// SIMATIC S7-200 project (STEP 7-Micro/WIN), CPU 224 REL 02.01

ORGANIZATION_BLOCK MAIN:OB1
TITLE=PROGRAM COMMENTS
BEGIN
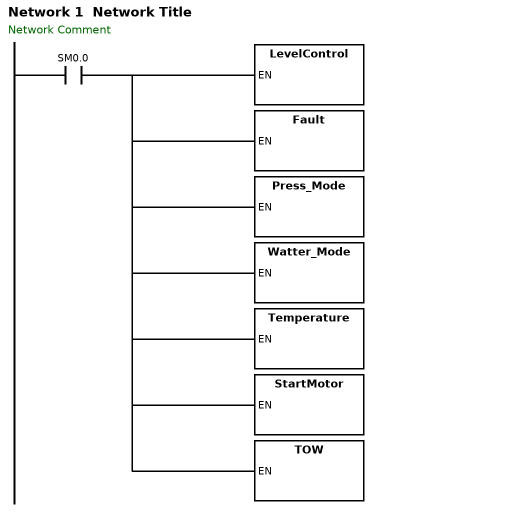
Network 1 // Network Title
// Network Comment
LD     SM0.0
CALL   LevelControl:SBR0
CALL   Fault:SBR1
CALL   Press_Mode:SBR2
CALL   Watter_Mode:SBR3
CALL   Temperature:SBR4
CALL   StartMotor:SBR5
CALL   TOW:SBR6
END_ORGANIZATION_BLOCK

SUBROUTINE_BLOCK LevelControl:SBR0
TITLE=SUBROUTINE COMMENTS
BEGIN
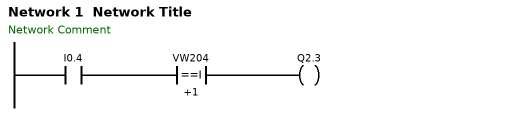
Network 1 // Network Title
// Network Comment
LD     I0.4
AW=    VW204, +1
=      Q2.3
END_SUBROUTINE_BLOCK

SUBROUTINE_BLOCK Fault:SBR1
TITLE=
BEGIN
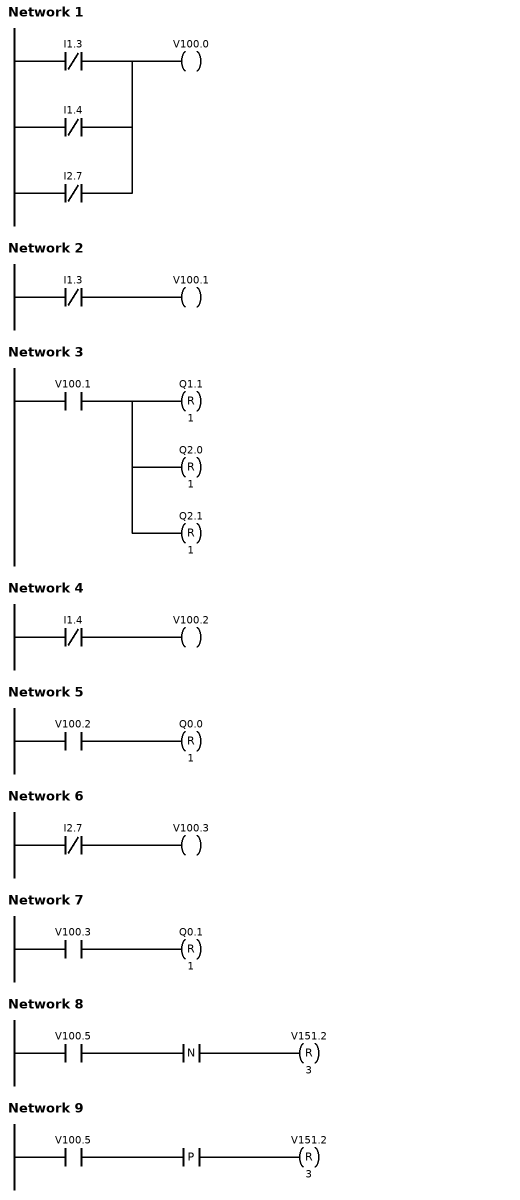
Network 1
LDN    I1.3
ON     I1.4
ON     I2.7
=      V100.0
Network 2
LDN    I1.3
=      V100.1
Network 3
LD     V100.1
R      Q1.1, 1
R      Q2.0, 1
R      Q2.1, 1
Network 4
LDN    I1.4
=      V100.2
Network 5
LD     V100.2
R      Q0.0, 1
Network 6
LDN    I2.7
=      V100.3
Network 7
LD     V100.3
R      Q0.1, 1
Network 8
LD     V100.5
ED
R      V151.2, 3
Network 9
LD     V100.5
EU
R      V151.2, 3
END_SUBROUTINE_BLOCK

SUBROUTINE_BLOCK Press_Mode:SBR2
TITLE=
BEGIN
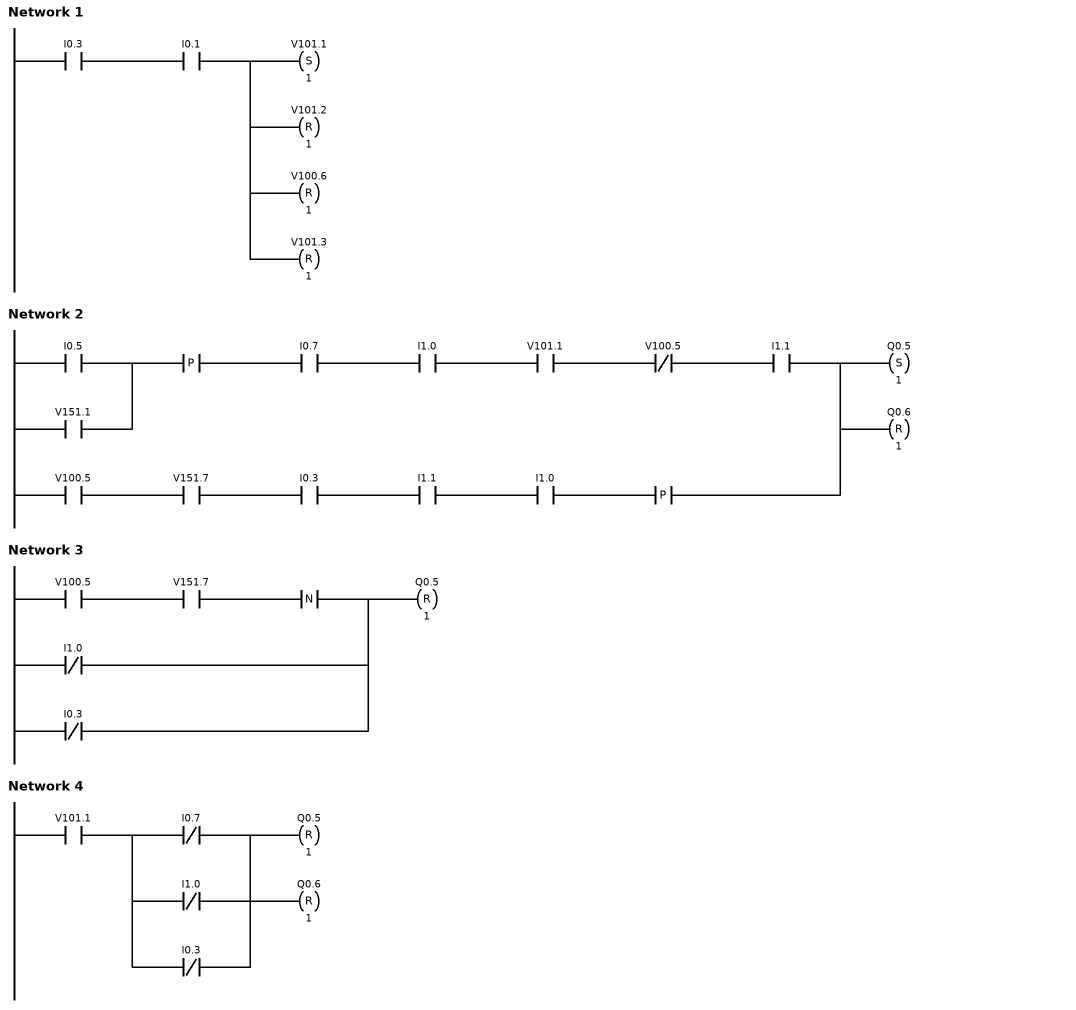
Network 1
LD     I0.3
A      I0.1
S      V101.1, 1
R      V101.2, 1
R      V100.6, 1
R      V101.3, 1
Network 2
LD     I0.5
O      V151.1
EU
A      I0.7
A      I1.0
A      V101.1
AN     V100.5
A      I1.1
LD     V100.5
A      V151.7
A      I0.3
A      I1.1
A      I1.0
EU
OLD
S      Q0.5, 1
R      Q0.6, 1
Network 3
LD     V100.5
A      V151.7
ED
ON     I1.0
ON     I0.3
R      Q0.5, 1
Network 4
LD     V101.1
LDN    I0.7
ON     I1.0
ON     I0.3
ALD
R      Q0.5, 1
R      Q0.6, 1
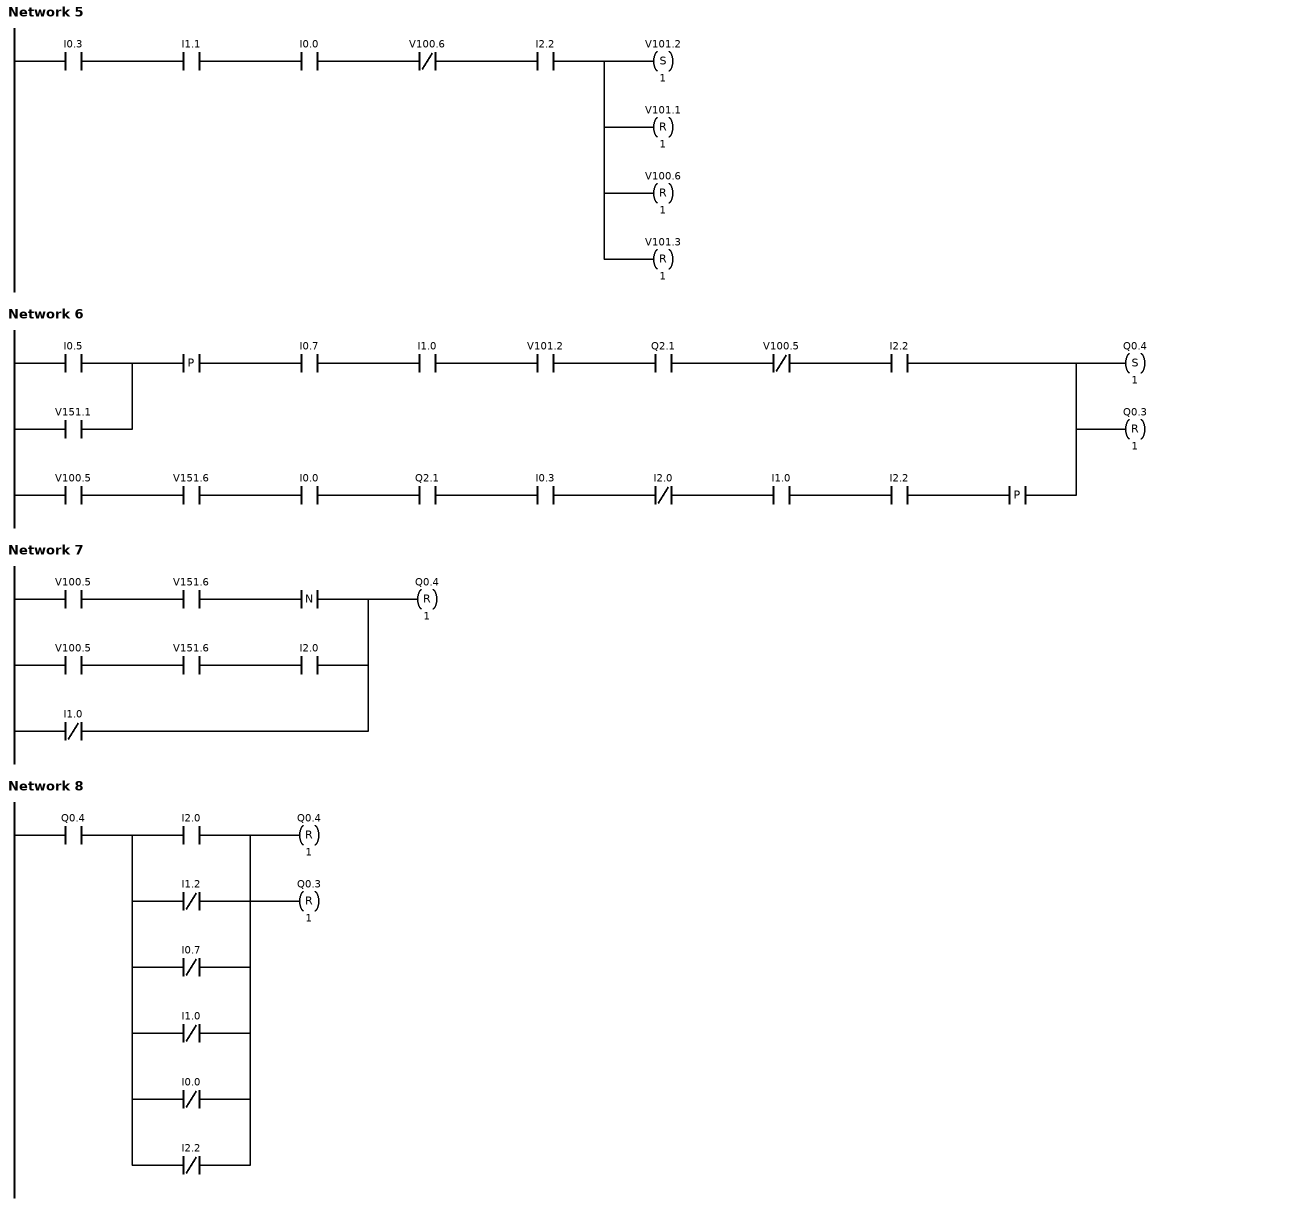
Network 5
LD     I0.3
A      I1.1
A      I0.0
AN     V100.6
A      I2.2
S      V101.2, 1
R      V101.1, 1
R      V100.6, 1
R      V101.3, 1
Network 6
LD     I0.5
O      V151.1
EU
A      I0.7
A      I1.0
A      V101.2
A      Q2.1
AN     V100.5
A      I2.2
LD     V100.5
A      V151.6
A      I0.0
A      Q2.1
A      I0.3
AN     I2.0
A      I1.0
A      I2.2
EU
OLD
S      Q0.4, 1
R      Q0.3, 1
Network 7
LD     V100.5
A      V151.6
ED
LD     V100.5
A      V151.6
A      I2.0
OLD
ON     I1.0
R      Q0.4, 1
Network 8
LD     Q0.4
LD     I2.0
ON     I1.2
ON     I0.7
ON     I1.0
ON     I0.0
ON     I2.2
ALD
R      Q0.4, 1
R      Q0.3, 1
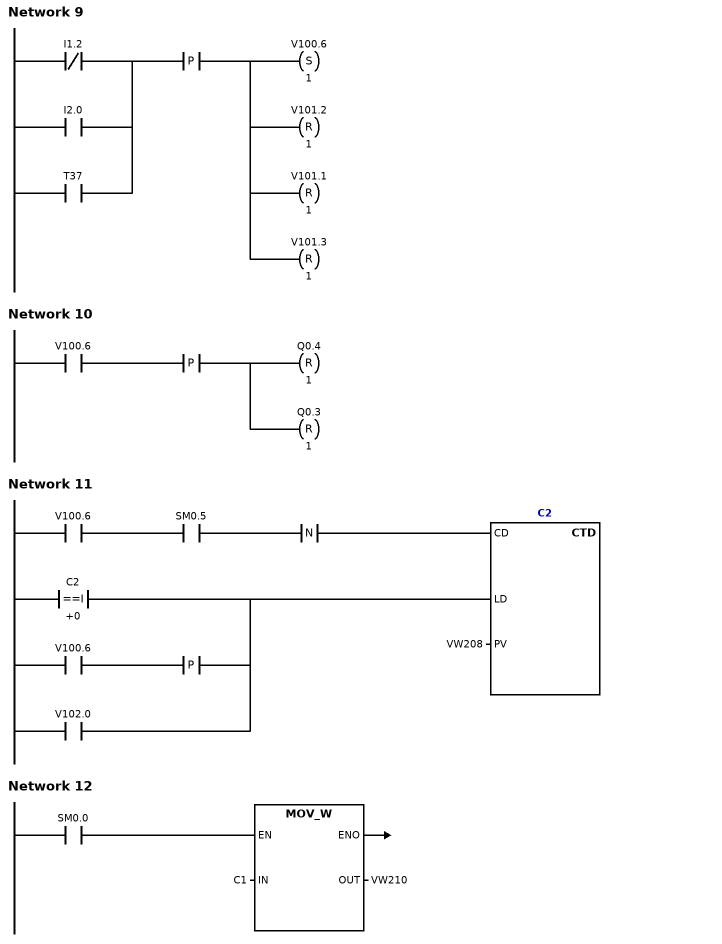
Network 9
LDN    I1.2
O      I2.0
O      T37
EU
S      V100.6, 1
R      V101.2, 1
R      V101.1, 1
R      V101.3, 1
Network 10
LD     V100.6
EU
R      Q0.4, 1
R      Q0.3, 1
Network 11
LD     V100.6
A      SM0.5
ED
LDW=   C2, +0
LD     V100.6
EU
OLD
O      V102.0
CTD    C2, VW208
Network 12
LD     SM0.0
MOVW   C1, VW210
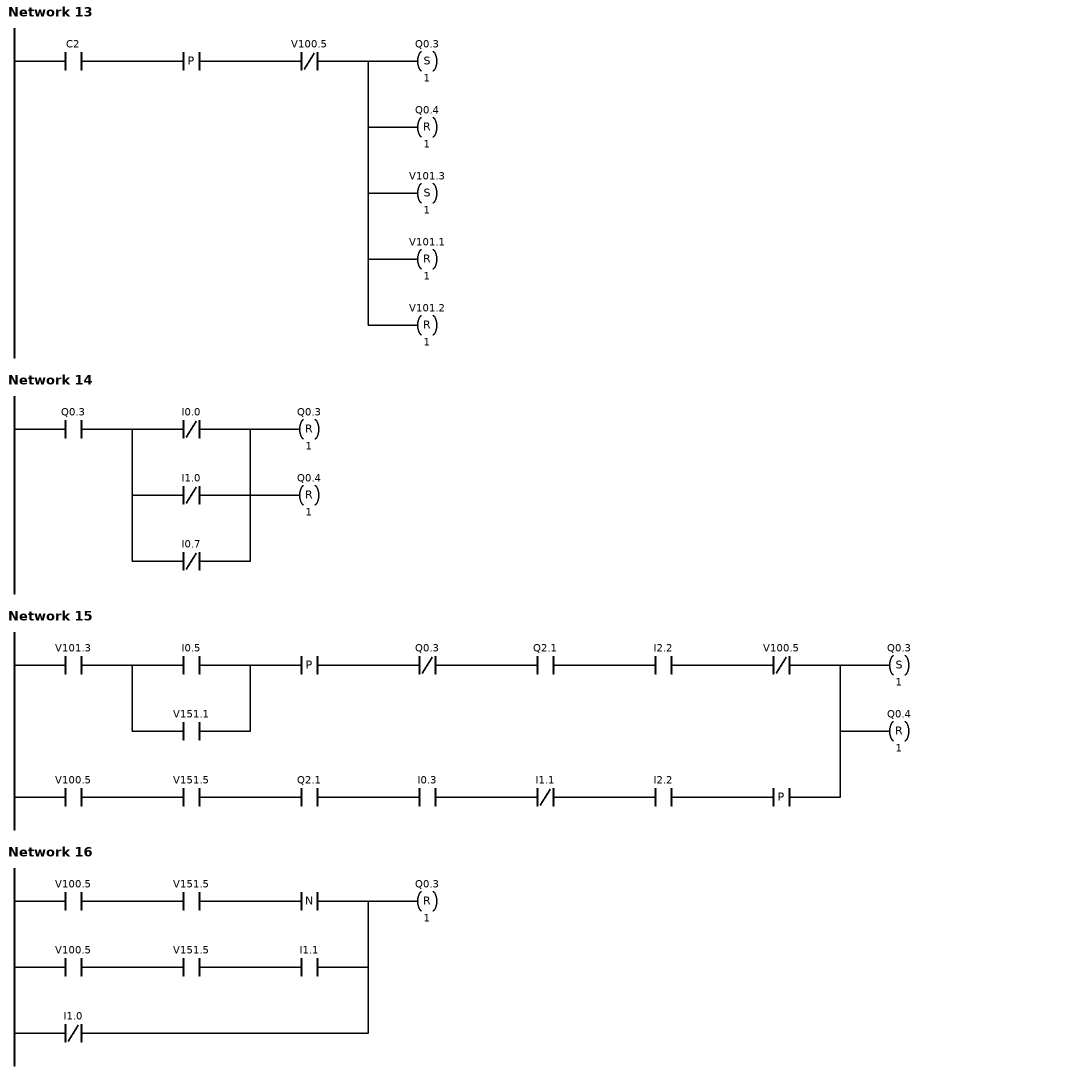
Network 13
LD     C2
EU
AN     V100.5
S      Q0.3, 1
R      Q0.4, 1
S      V101.3, 1
R      V101.1, 1
R      V101.2, 1
Network 14
LD     Q0.3
LDN    I0.0
ON     I1.0
ON     I0.7
ALD
R      Q0.3, 1
R      Q0.4, 1
Network 15
LD     V101.3
LD     I0.5
O      V151.1
ALD
EU
AN     Q0.3
A      Q2.1
A      I2.2
AN     V100.5
LD     V100.5
A      V151.5
A      Q2.1
A      I0.3
AN     I1.1
A      I2.2
EU
OLD
S      Q0.3, 1
R      Q0.4, 1
Network 16
LD     V100.5
A      V151.5
ED
LD     V100.5
A      V151.5
A      I1.1
OLD
ON     I1.0
R      Q0.3, 1
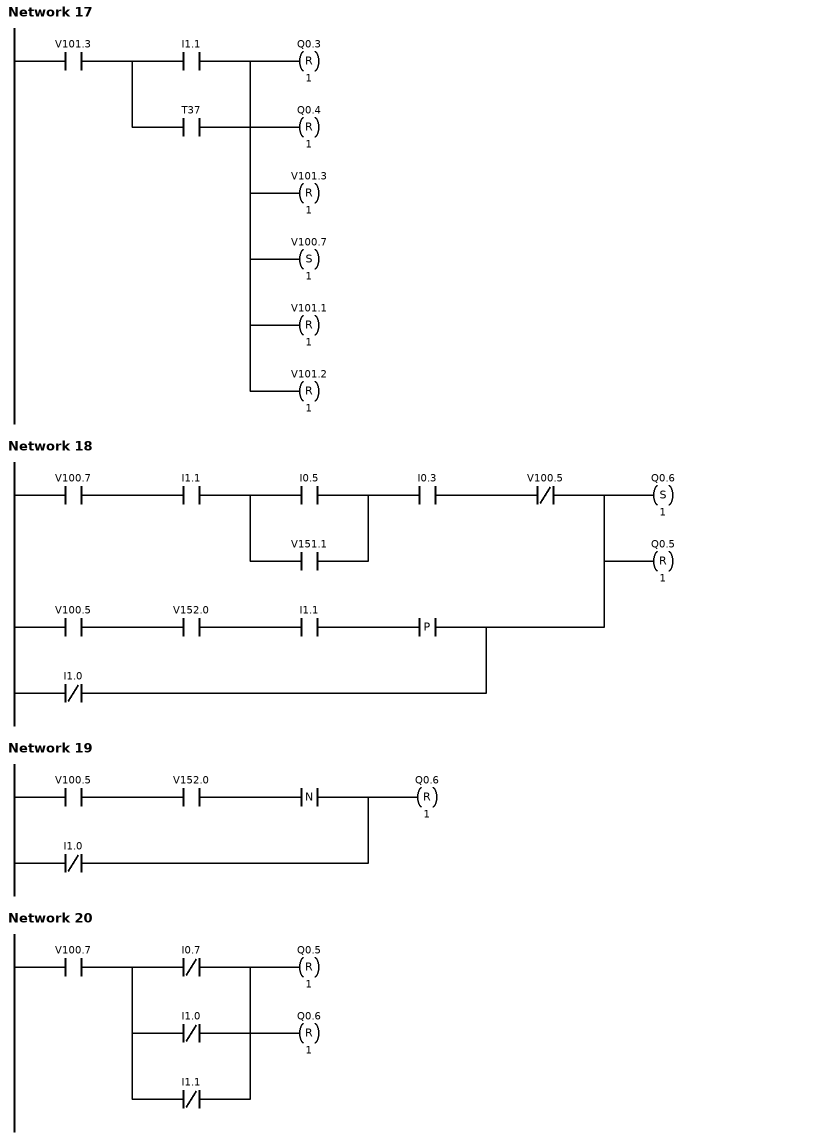
Network 17
LD     V101.3
LD     I1.1
O      T37
ALD
R      Q0.3, 1
R      Q0.4, 1
R      V101.3, 1
S      V100.7, 1
R      V101.1, 1
R      V101.2, 1
Network 18
LD     V100.7
A      I1.1
LD     I0.5
O      V151.1
ALD
A      I0.3
AN     V100.5
LD     V100.5
A      V152.0
A      I1.1
EU
ON     I1.0
OLD
S      Q0.6, 1
R      Q0.5, 1
Network 19
LD     V100.5
A      V152.0
ED
ON     I1.0
R      Q0.6, 1
Network 20
LD     V100.7
LDN    I0.7
ON     I1.0
ON     I1.1
ALD
R      Q0.5, 1
R      Q0.6, 1
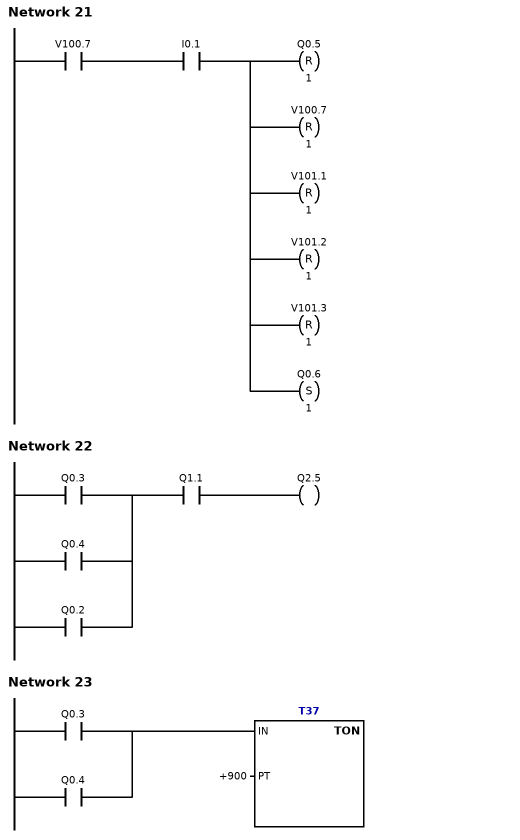
Network 21
LD     V100.7
A      I0.1
R      Q0.5, 1
R      V100.7, 1
R      V101.1, 1
R      V101.2, 1
R      V101.3, 1
S      Q0.6, 1
Network 22
LD     Q0.3
O      Q0.4
O      Q0.2
A      Q1.1
=      Q2.5
Network 23
LD     Q0.3
O      Q0.4
TON    T37, +900
END_SUBROUTINE_BLOCK

SUBROUTINE_BLOCK Watter_Mode:SBR3
TITLE=
BEGIN
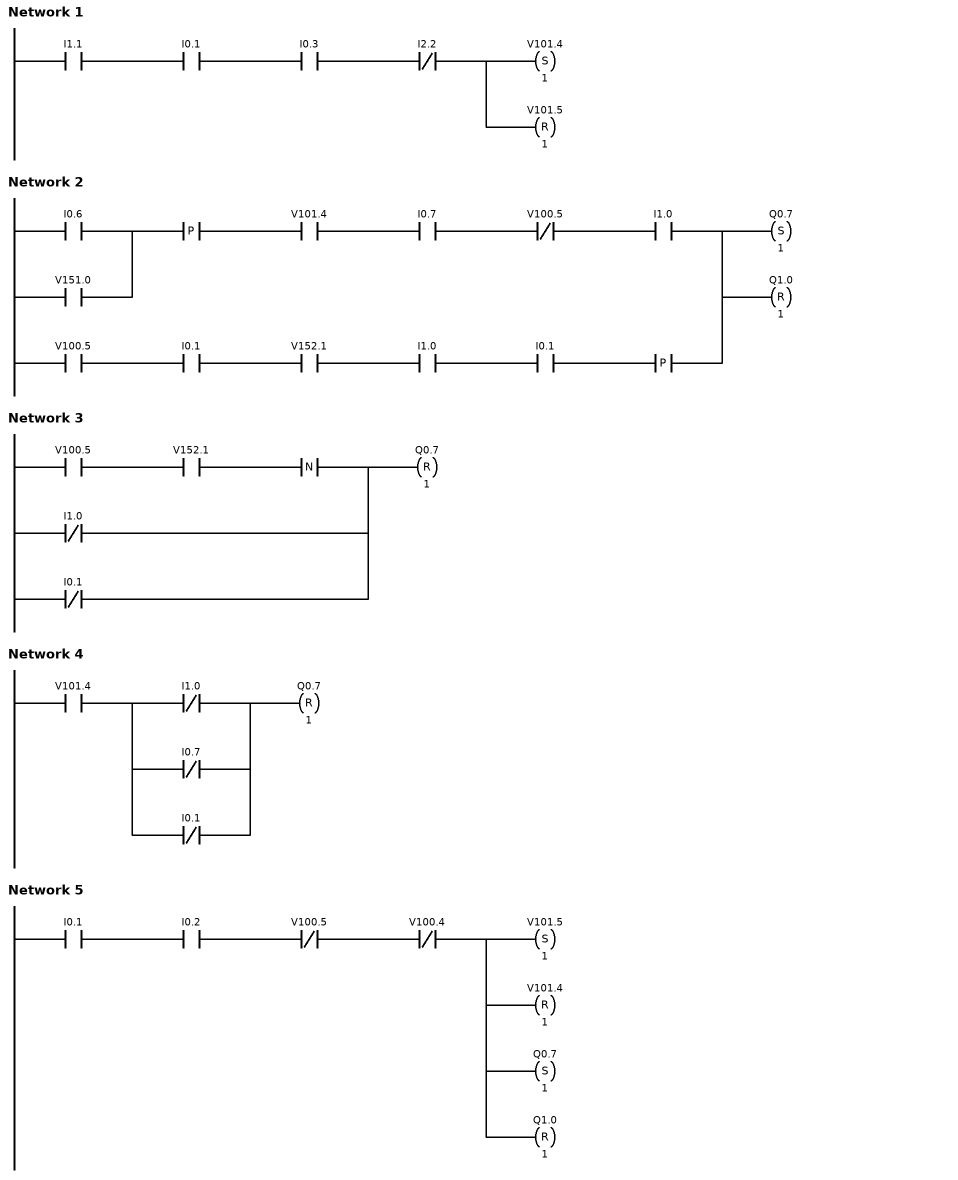
Network 1
LD     I1.1
A      I0.1
A      I0.3
AN     I2.2
S      V101.4, 1
R      V101.5, 1
Network 2
LD     I0.6
O      V151.0
EU
A      V101.4
A      I0.7
AN     V100.5
A      I1.0
LD     V100.5
A      I0.1
A      V152.1
A      I1.0
A      I0.1
EU
OLD
S      Q0.7, 1
R      Q1.0, 1
Network 3
LD     V100.5
A      V152.1
ED
ON     I1.0
ON     I0.1
R      Q0.7, 1
Network 4
LD     V101.4
LDN    I1.0
ON     I0.7
ON     I0.1
ALD
R      Q0.7, 1
Network 5
LD     I0.1
A      I0.2
AN     V100.5
AN     V100.4
S      V101.5, 1
R      V101.4, 1
S      Q0.7, 1
R      Q1.0, 1
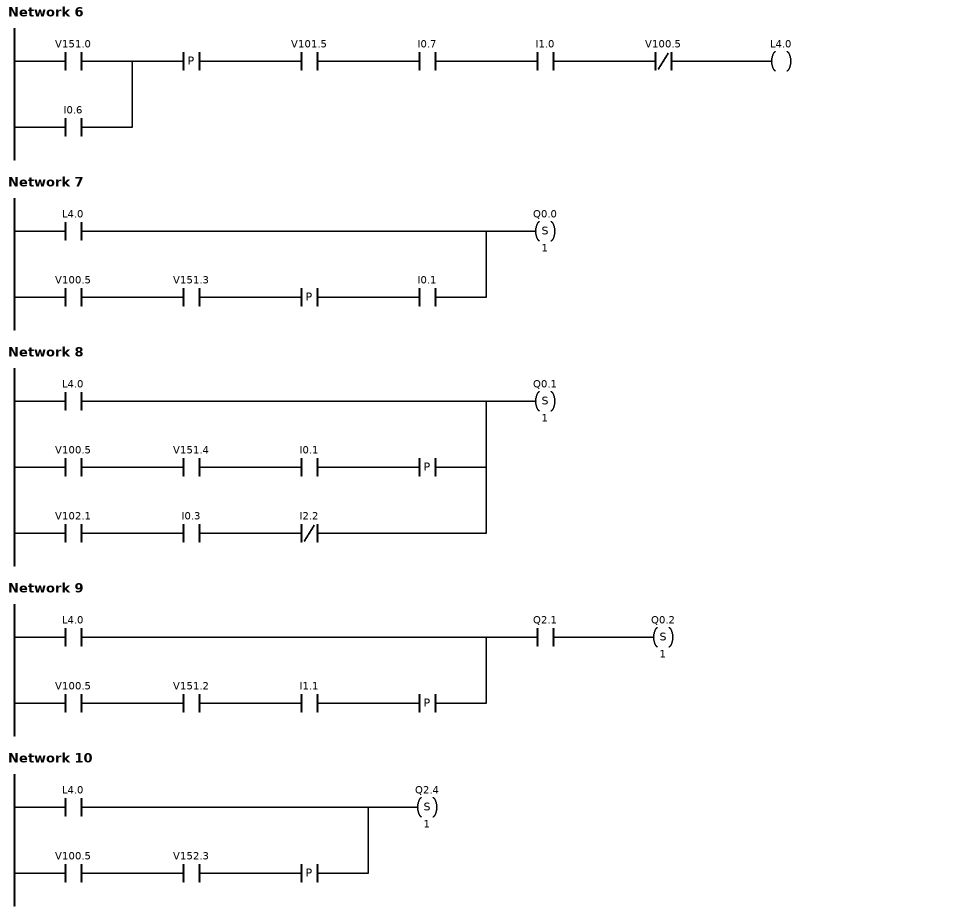
Network 6
LD     V151.0
O      I0.6
EU
A      V101.5
A      I0.7
A      I1.0
AN     V100.5
=      L4.0
Network 7
LD     L4.0
LD     V100.5
A      V151.3
EU
A      I0.1
OLD
S      Q0.0, 1
Network 8
LD     L4.0
LD     V100.5
A      V151.4
A      I0.1
EU
OLD
LD     V102.1
A      I0.3
AN     I2.2
OLD
S      Q0.1, 1
Network 9
LD     L4.0
LD     V100.5
A      V151.2
A      I1.1
EU
OLD
A      Q2.1
S      Q0.2, 1
Network 10
LD     L4.0
LD     V100.5
A      V152.3
EU
OLD
S      Q2.4, 1
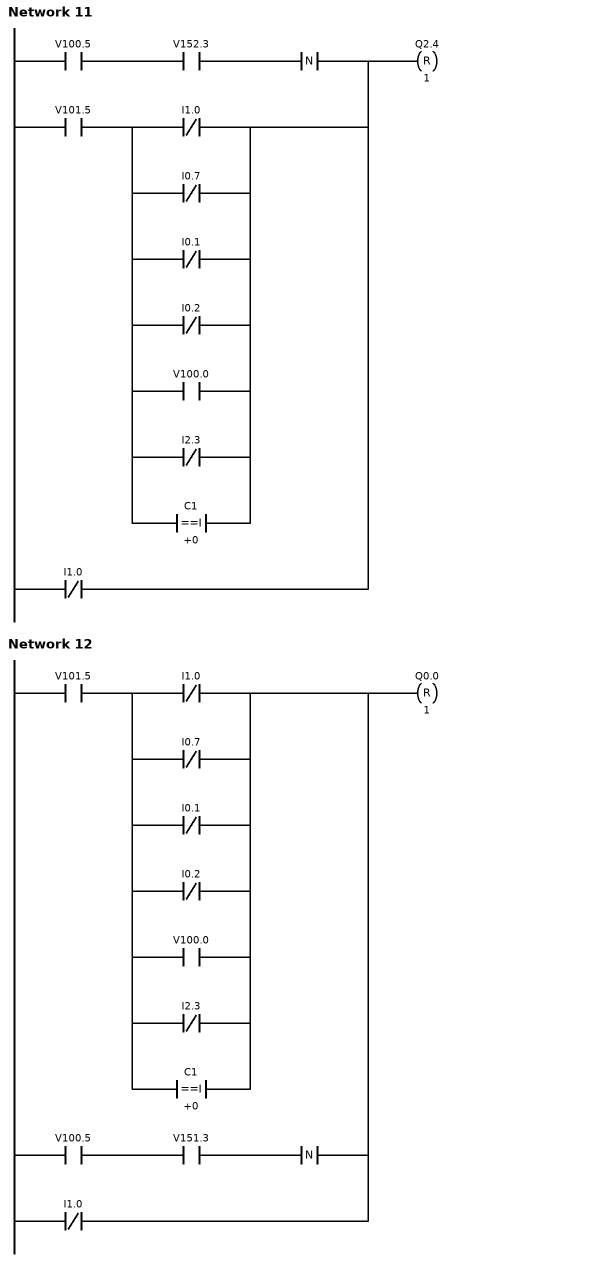
Network 11
LD     V100.5
A      V152.3
ED
LD     V101.5
LDN    I1.0
ON     I0.7
ON     I0.1
ON     I0.2
O      V100.0
ON     I2.3
OW=    C1, +0
ALD
OLD
ON     I1.0
R      Q2.4, 1
Network 12
LD     V101.5
LDN    I1.0
ON     I0.7
ON     I0.1
ON     I0.2
O      V100.0
ON     I2.3
OW=    C1, +0
ALD
LD     V100.5
A      V151.3
ED
ON     I1.0
OLD
R      Q0.0, 1
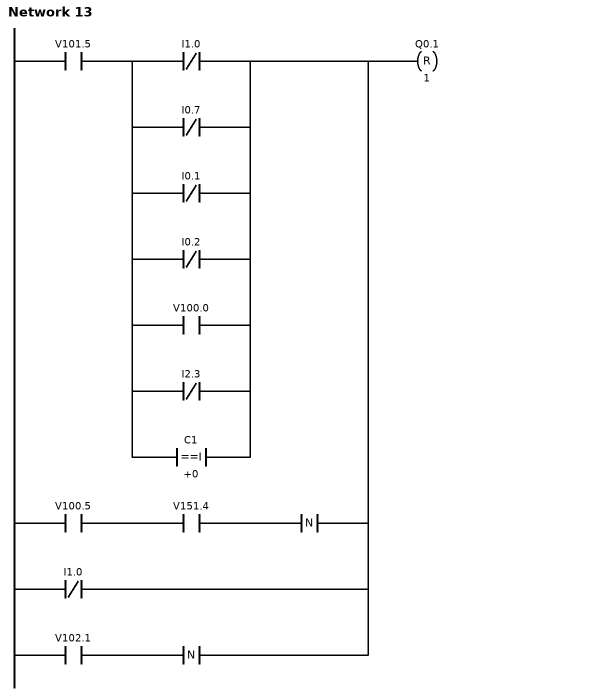
Network 13
LD     V101.5
LDN    I1.0
ON     I0.7
ON     I0.1
ON     I0.2
O      V100.0
ON     I2.3
OW=    C1, +0
ALD
LD     V100.5
A      V151.4
ED
ON     I1.0
LD     V102.1
ED
OLD
OLD
R      Q0.1, 1
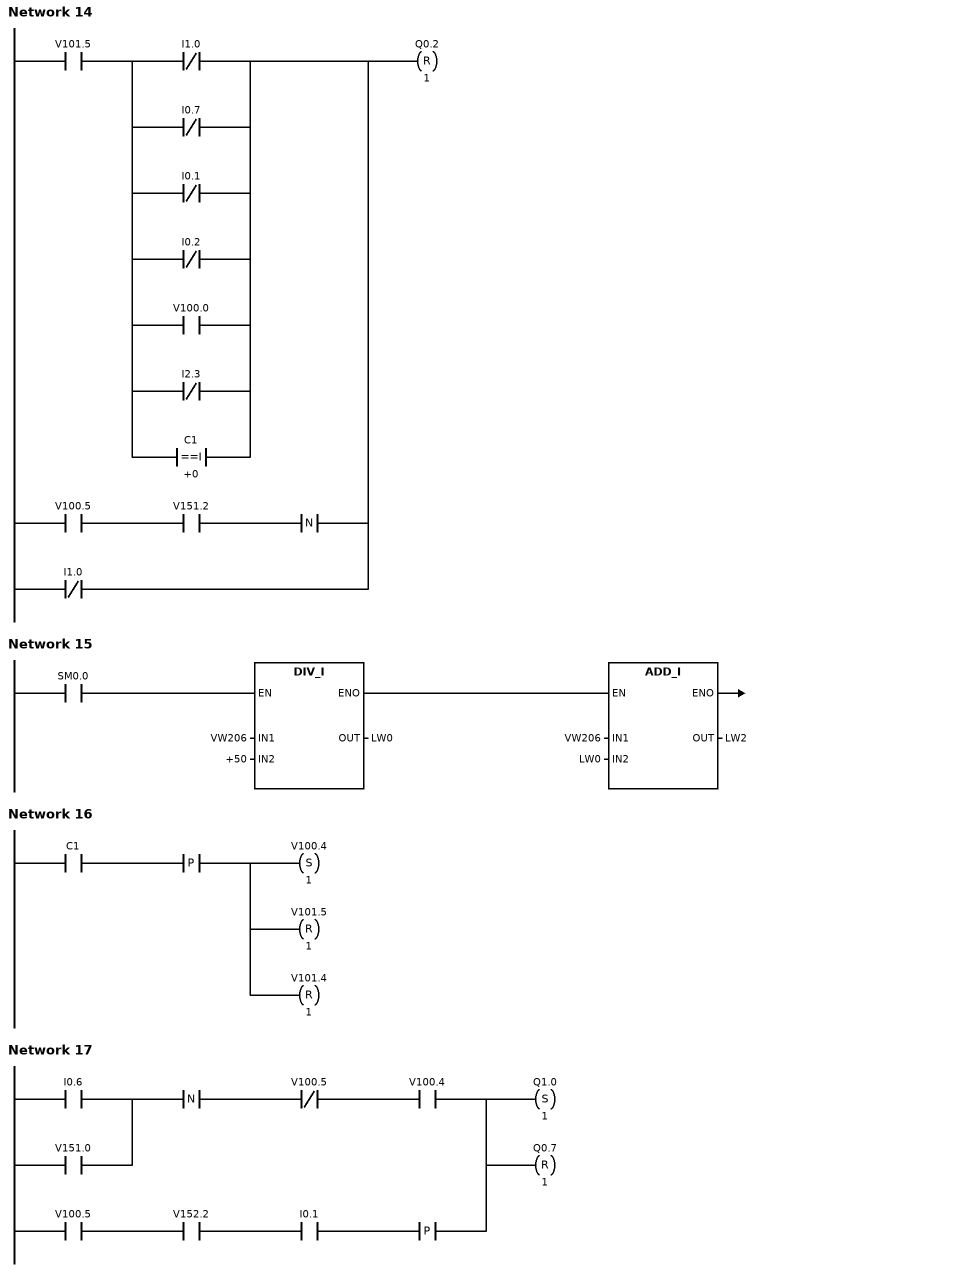
Network 14
LD     V101.5
LDN    I1.0
ON     I0.7
ON     I0.1
ON     I0.2
O      V100.0
ON     I2.3
OW=    C1, +0
ALD
LD     V100.5
A      V151.2
ED
ON     I1.0
OLD
R      Q0.2, 1
Network 15
LD     SM0.0
MOVW   VW206, LW0
AENO
/I     +50, LW0
AENO
MOVW   VW206, LW2
+I     LW0, LW2
Network 16
LD     C1
EU
S      V100.4, 1
R      V101.5, 1
R      V101.4, 1
Network 17
LD     I0.6
O      V151.0
ED
AN     V100.5
A      V100.4
LD     V100.5
A      V152.2
A      I0.1
EU
OLD
S      Q1.0, 1
R      Q0.7, 1
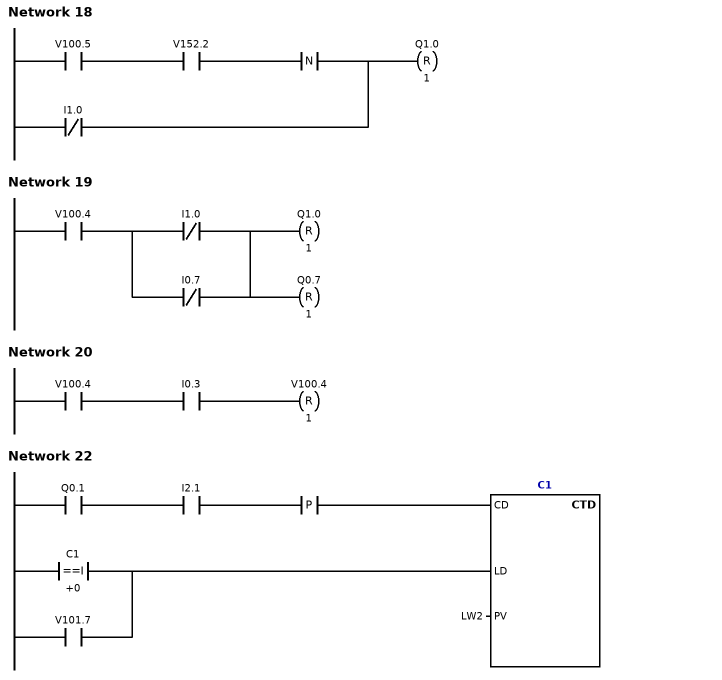
Network 18
LD     V100.5
A      V152.2
ED
ON     I1.0
R      Q1.0, 1
Network 19
LD     V100.4
LDN    I1.0
ON     I0.7
ALD
R      Q1.0, 1
R      Q0.7, 1
Network 20
LD     V100.4
A      I0.3
R      V100.4, 1
Network 22
LD     Q0.1
A      I2.1
EU
LDW=   C1, +0
O      V101.7
CTD    C1, LW2
END_SUBROUTINE_BLOCK

SUBROUTINE_BLOCK Temperature:SBR4
TITLE=
BEGIN
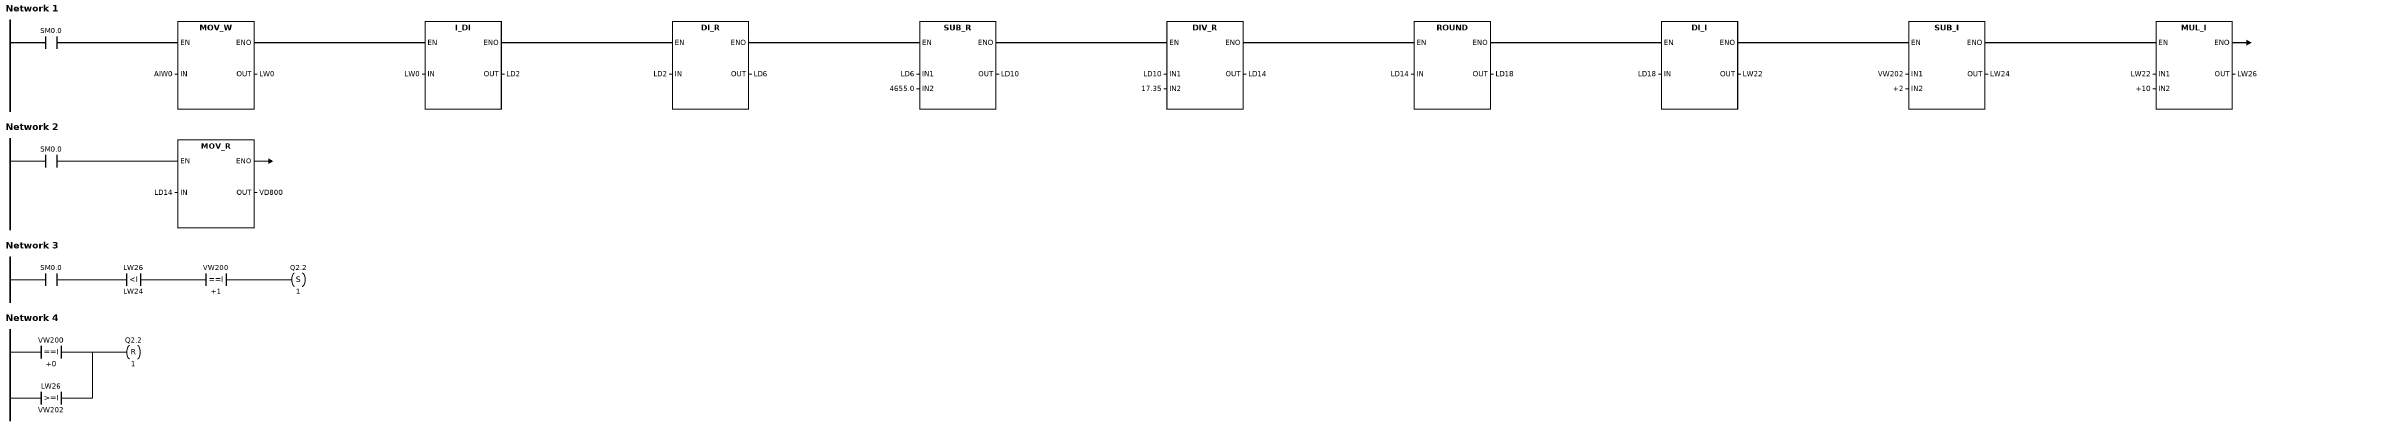
Network 1
LD     SM0.0
MOVW   AIW0, LW0
AENO
ITD    LW0, LD2
AENO
DTR    LD2, LD6
AENO
MOVR   LD6, LD10
AENO
-R     4655.0, LD10
AENO
MOVR   LD10, LD14
AENO
/R     17.35, LD14
AENO
ROUND  LD14, LD18
AENO
DTI    LD18, LW22
AENO
MOVW   VW202, LW24
AENO
-I     +2, LW24
AENO
MOVW   LW22, LW26
*I     +10, LW26
Network 2
LD     SM0.0
MOVR   LD14, VD800
Network 3
LD     SM0.0
AW<    LW26, LW24
AW=    VW200, +1
S      Q2.2, 1
Network 4
LDW=   VW200, +0
OW>=   LW26, VW202
R      Q2.2, 1
END_SUBROUTINE_BLOCK

SUBROUTINE_BLOCK StartMotor:SBR5
TITLE=
BEGIN
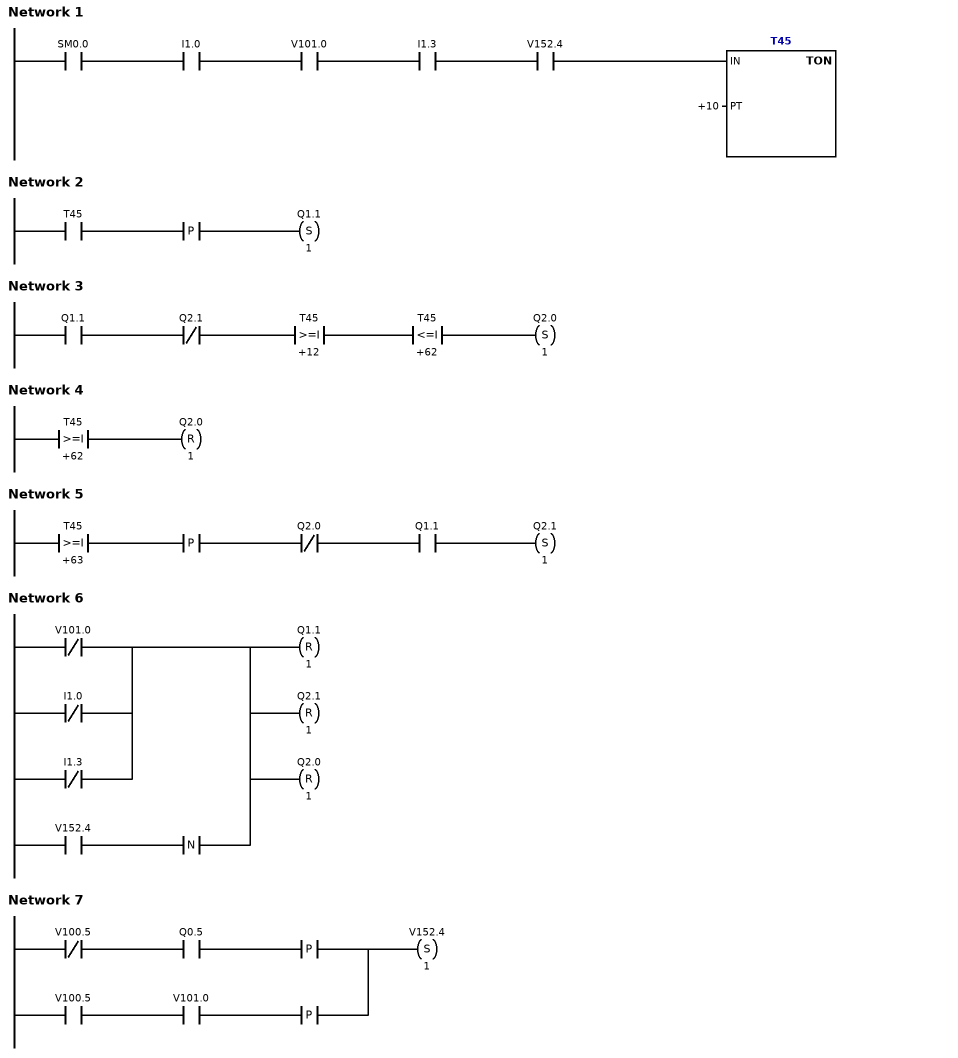
Network 1
LD     SM0.0
A      I1.0
A      V101.0
A      I1.3
A      V152.4
TON    T45, +10
Network 2
LD     T45
EU
S      Q1.1, 1
Network 3
LD     Q1.1
AN     Q2.1
AW>=   T45, +12
AW<=   T45, +62
S      Q2.0, 1
Network 4
LDW>=  T45, +62
R      Q2.0, 1
Network 5
LDW>=  T45, +63
EU
AN     Q2.0
A      Q1.1
S      Q2.1, 1
Network 6
LDN    V101.0
ON     I1.0
ON     I1.3
LD     V152.4
ED
OLD
R      Q1.1, 1
R      Q2.1, 1
R      Q2.0, 1
Network 7
LDN    V100.5
A      Q0.5
EU
LD     V100.5
A      V101.0
EU
OLD
S      V152.4, 1
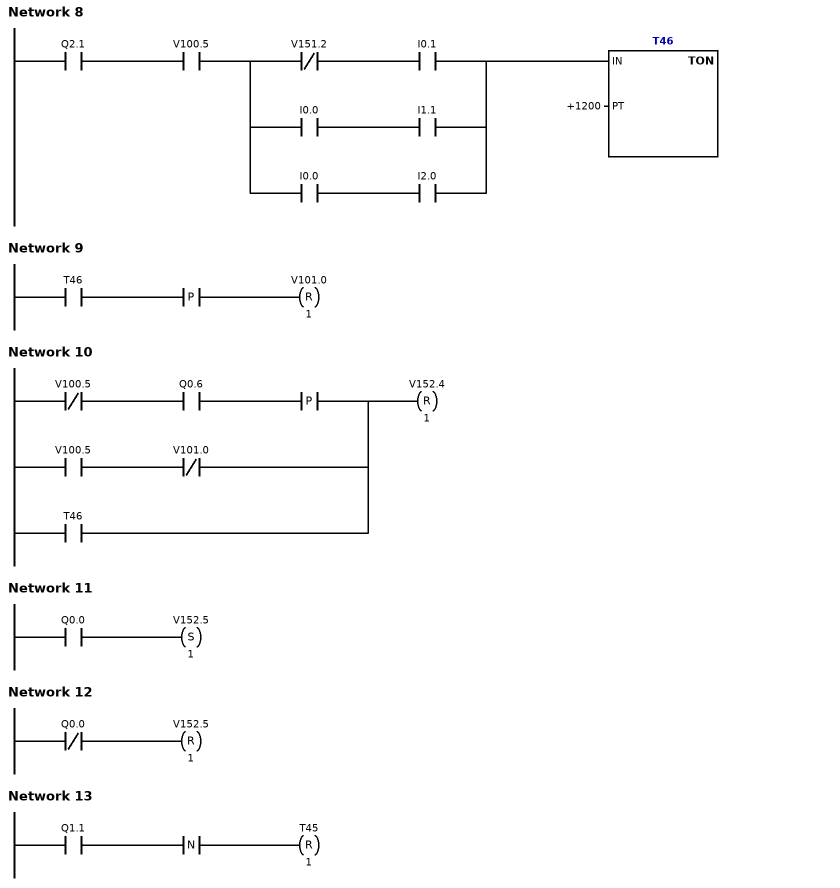
Network 8
LD     Q2.1
A      V100.5
LDN    V151.2
A      I0.1
LD     I0.0
A      I1.1
OLD
LD     I0.0
A      I2.0
OLD
ALD
TON    T46, +1200
Network 9
LD     T46
EU
R      V101.0, 1
Network 10
LDN    V100.5
A      Q0.6
EU
LD     V100.5
AN     V101.0
OLD
O      T46
R      V152.4, 1
Network 11
LD     Q0.0
S      V152.5, 1
Network 12
LDN    Q0.0
R      V152.5, 1
Network 13
LD     Q1.1
ED
R      T45, 1
END_SUBROUTINE_BLOCK

SUBROUTINE_BLOCK TOW:SBR6
TITLE=
BEGIN
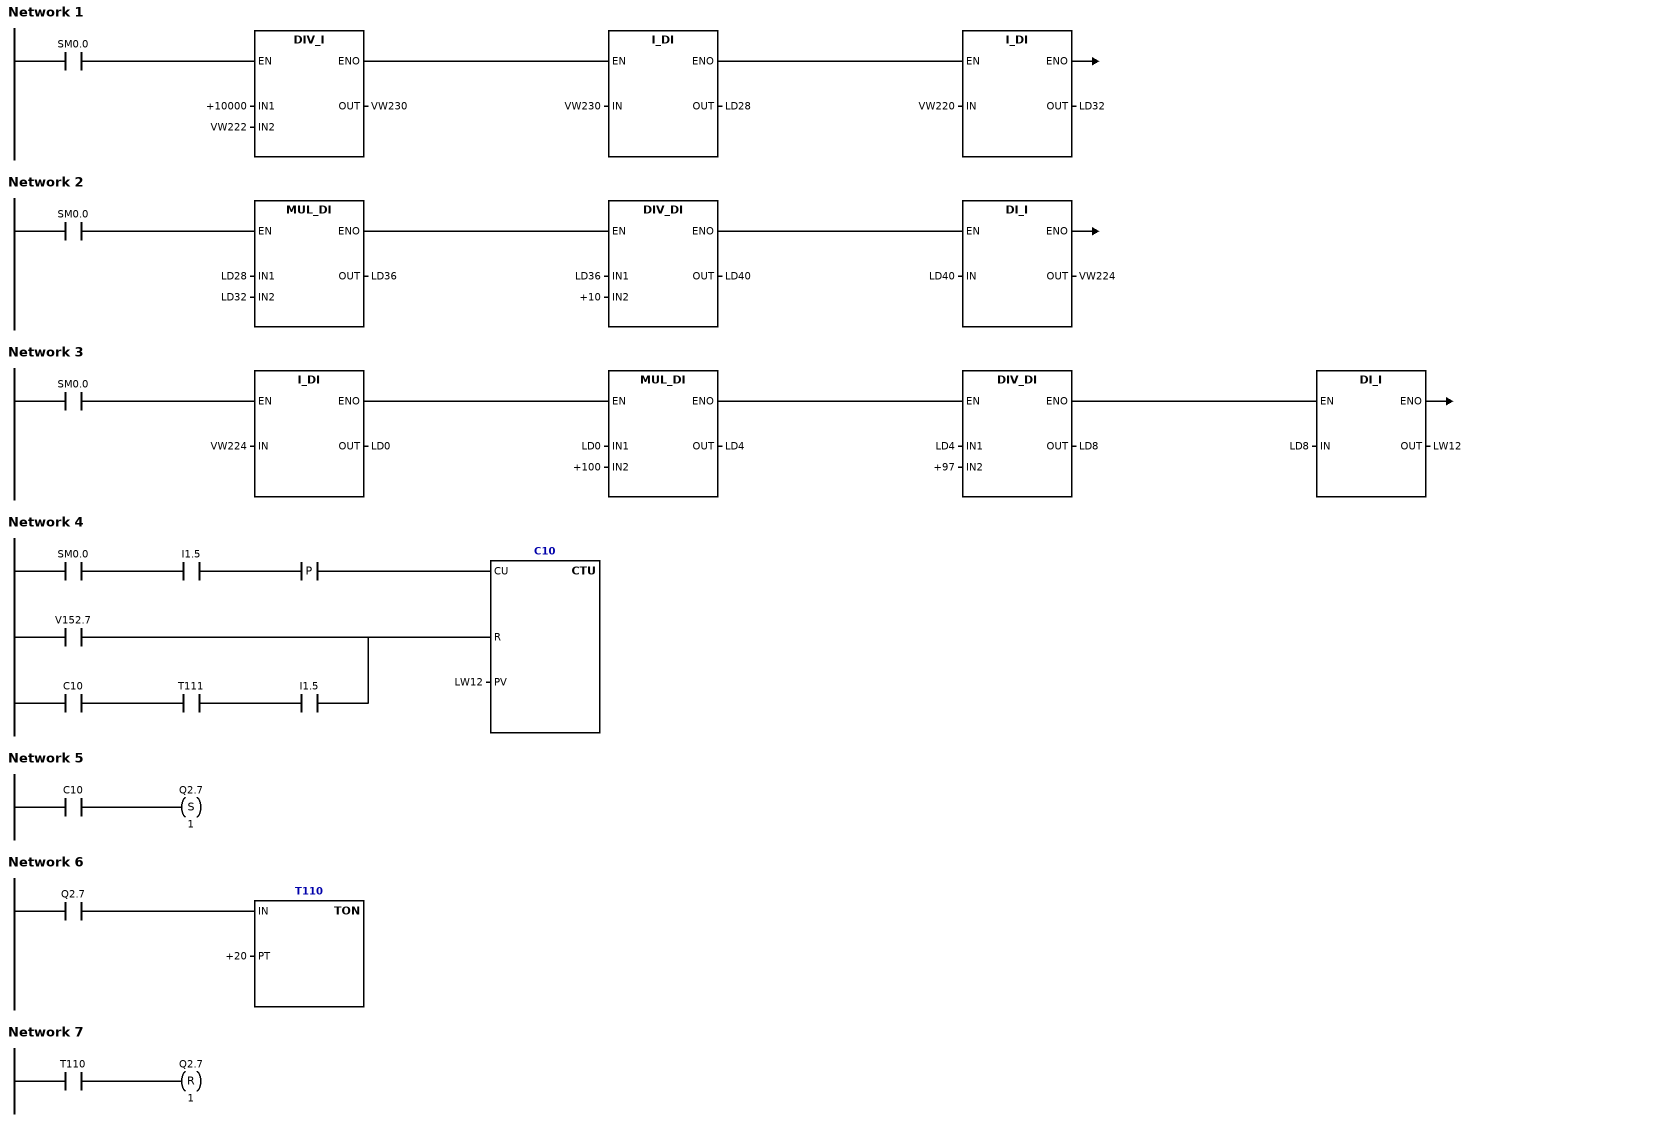
Network 1
LD     SM0.0
MOVW   +10000, VW230
AENO
/I     VW222, VW230
AENO
ITD    VW230, LD28
AENO
ITD    VW220, LD32
Network 2
LD     SM0.0
MOVD   LD28, LD36
AENO
*D     LD32, LD36
AENO
MOVD   LD36, LD40
AENO
/D     +10, LD40
AENO
DTI    LD40, VW224
Network 3
LD     SM0.0
ITD    VW224, LD0
AENO
MOVD   LD0, LD4
AENO
*D     +100, LD4
AENO
MOVD   LD4, LD8
AENO
/D     +97, LD8
AENO
DTI    LD8, LW12
Network 4
LD     SM0.0
A      I1.5
EU
LD     V152.7
LD     C10
A      T111
A      I1.5
OLD
CTU    C10, LW12
Network 5
LD     C10
S      Q2.7, 1
Network 6
LD     Q2.7
TON    T110, +20
Network 7
LD     T110
R      Q2.7, 1
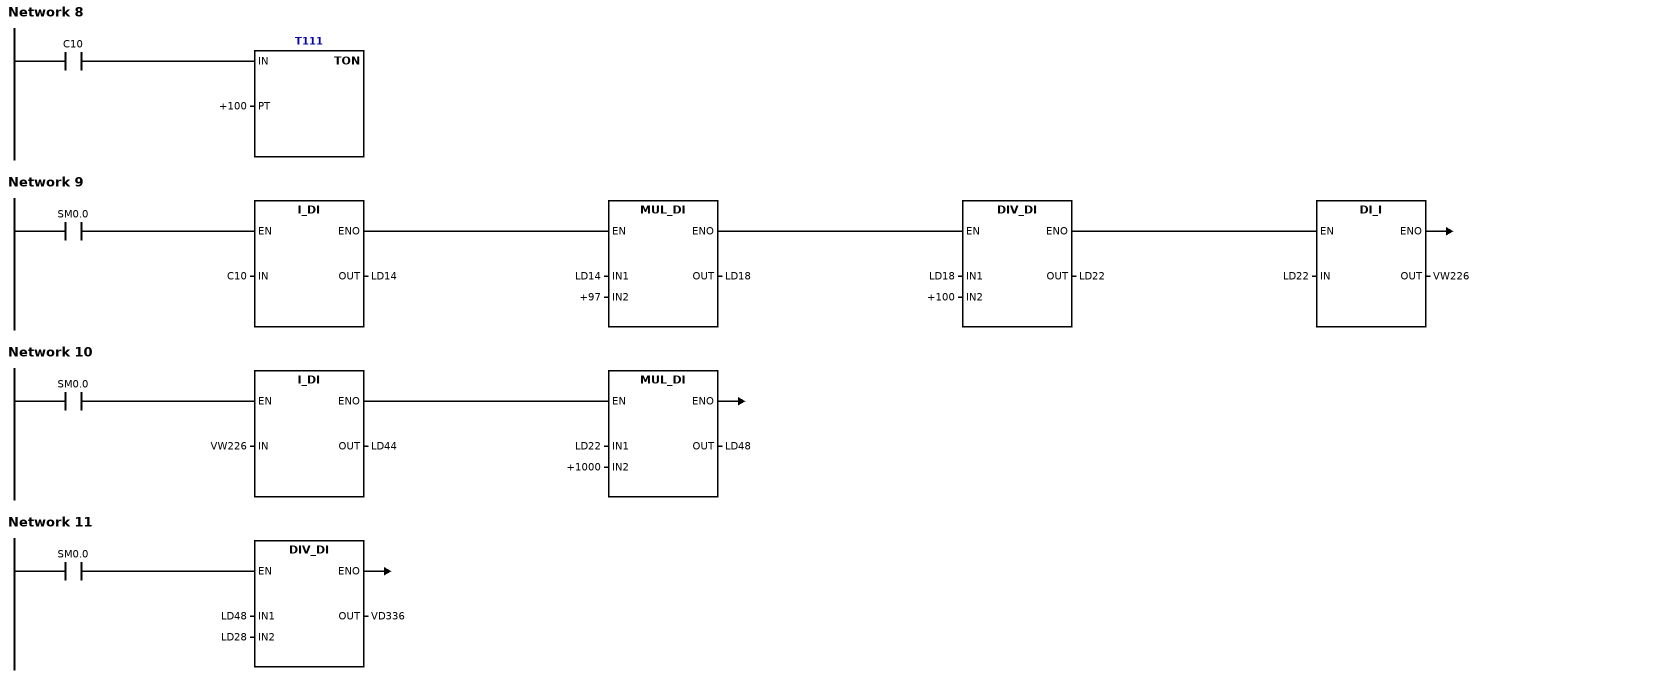
Network 8
LD     C10
TON    T111, +100
Network 9
LD     SM0.0
ITD    C10, LD14
AENO
MOVD   LD14, LD18
AENO
*D     +97, LD18
AENO
MOVD   LD18, LD22
AENO
/D     +100, LD22
AENO
DTI    LD22, VW226
Network 10
LD     SM0.0
ITD    VW226, LD44
AENO
MOVD   LD22, LD48
*D     +1000, LD48
Network 11
LD     SM0.0
MOVD   LD48, VD336
/D     LD28, VD336
END_SUBROUTINE_BLOCK
